TEXTLIST EL1809_S_2
  1 = 'SubInkTankLevel P2' | chinese: '二级墨盒液位图层2' | Chinese: '二级墨盒液位图层2'
  2 = 'SubInkTankLevel W1' | chinese: '二级墨盒液位W1' | Chinese: '二级墨盒液位W1'
  3 = 'SubInkTankLevel W2' | chinese: '二级墨盒液位W2' | Chinese: '二级墨盒液位W2'
  4 = 'SubInkTankLevel W3' | chinese: '二级墨盒液位W3' | Chinese: '二级墨盒液位W3'
  5 = 'SubInkTankLevel W4' | chinese: '二级墨盒液位W4' | Chinese: '二级墨盒液位W4'
  6 = 'ProtectTankLevel_C' | chinese: '真空保护瓶液位1' | Chinese: '真空保护瓶液位1'
  7 = 'ProtectTankLevel_W' | chinese: '真空保护瓶液位2' | Chinese: '真空保护瓶液位2'
  8 = 'Purge button' | chinese: '正压按钮' | Chinese: '正压按钮'
  9 = 'Color vac button' | chinese: '彩色正负压切换按钮' | Chinese: '彩色正负压切换按钮'
  10 = 'White vac button' | chinese: '白色正负压切换按钮' | Chinese: '白色正负压切换按钮'
  11 = ''
  12 = ''
  13 = ''
  14 = ''
  15 = ''
  16 = ''
   = ''
END_TEXTLIST

(* stored: Version 1.1.0.1, ProductVersion 3.1.4024.11
   TextList EL1809_S_2: Id {f249efbc-130d-46f8-bb7f-21243d9958b8} *)
